PROGRAM P2_06_Device_Ctrl
VAR
	
	fbDischargeValve				:FB_Valve53_Ctrl;	
	bDischargeOpen					:BOOL;
	bDischargeClose					:BOOL;

	fbMixer_Cmd						:FB_Mixer_Ctrl;
	fbMixerSpeed_Cmd				:FB_AnalogOutput;
	fbMixerSpeed_Cmd2				:FB_Scale;

	fChopper1_Cmd					:FB_Chopper_Ctrl;
	fChopper2_Cmd					:FB_Chopper_Ctrl;
	
	fbWater_V1020_Cmd				:FB_Valve_Ctrl;
	fbWarmWater_Cmd					:FB_Valve_Ctrl;
	fbColdWater_Cmd					:FB_Valve_Ctrl;
	fbProcessWater_V1025_Cmd		:FB_Valve_Ctrl;
	fbCleaningAir_V1030_Cmd			:FB_Valve_Ctrl;
	fbTightAir_V1100_Cmd			:FB_Valve_Ctrl;
	
	fbChopper1_Air_V1080_Cmd		:FB_Valve_Ctrl;
	fbChopper1_Water_V1580_Cmd		:FB_Valve_Ctrl;
	fbChopper1_Drain_V1150_Cmd		:FB_Valve_Ctrl;
	
	fbChopper2_Air_V1090_Cmd		:FB_Valve_Ctrl;
	fbChopper2_Water_V1570_Cmd		:FB_Valve_Ctrl;
	fbChopper2_Drain_V1160_Cmd		:FB_Valve_Ctrl;
	
	fbDrainSocket_V1010_Cmd			:FB_Valve_Ctrl;
	
	tonChopper2Delay				:TON;
	
	test		:BOOL;
	fbMixerSpeed_Cmd3: FB_Scale;
	TON_0: TON;
	TON_1: TON;
	TON_2: TON;
END_VAR

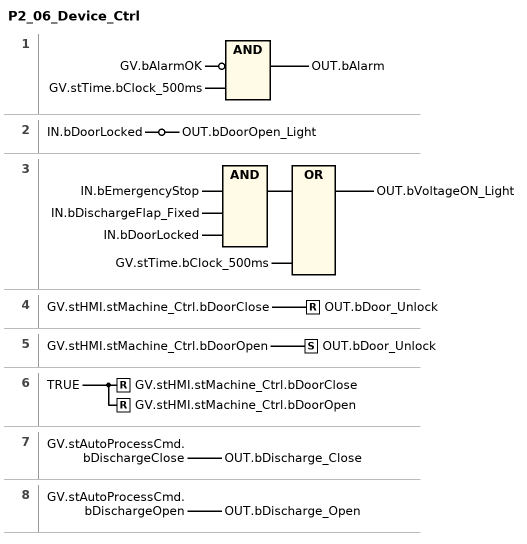
// NETWORK 1
OUT.bAlarm := NOT GV.bAlarmOK AND GV.stTime.bClock_500ms;

// NETWORK 2
OUT.bDoorOpen_Light := NOT IN.bDoorLocked;

// NETWORK 3
OUT.bVoltageON_Light := IN.bEmergencyStop AND IN.bDischargeFlap_Fixed AND IN.bDoorLocked OR GV.stTime.bClock_500ms;

// NETWORK 4
OUT.bDoor_Unlock R= GV.stHMI.stMachine_Ctrl.bDoorClose;

// NETWORK 5
OUT.bDoor_Unlock S= GV.stHMI.stMachine_Ctrl.bDoorOpen;

// NETWORK 6
GV.stHMI.stMachine_Ctrl.bDoorClose R= TRUE;
GV.stHMI.stMachine_Ctrl.bDoorOpen R= TRUE;

// NETWORK 7
OUT.bDischarge_Close := GV.stAutoProcessCmd.bDischargeClose;

// NETWORK 8
OUT.bDischarge_Open := GV.stAutoProcessCmd.bDischargeOpen;

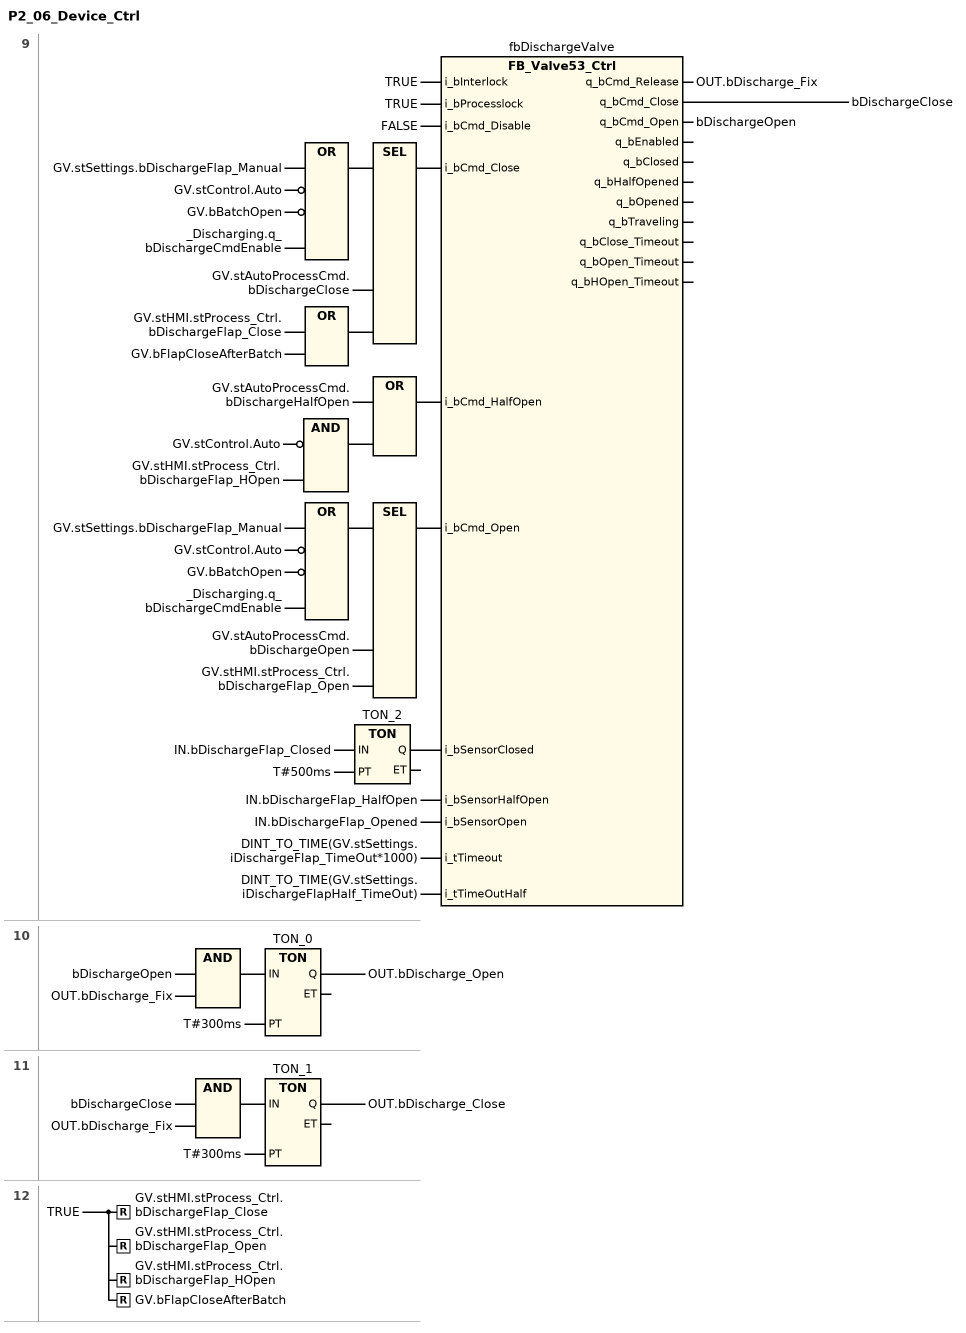
// NETWORK 9
TON_2(IN := IN.bDischargeFlap_Closed, PT := T#500ms); // TON
fbDischargeValve(
    i_bInterlock := TRUE,
    i_bProcesslock := TRUE,
    i_bCmd_Disable := FALSE,
    i_bCmd_Close := SEL(GV.stSettings.bDischargeFlap_Manual OR NOT GV.stControl.Auto OR NOT GV.bBatchOpen OR _Discharging.q_bDischargeCmdEnable, GV.stAutoProcessCmd.bDischargeClose, GV.stHMI.stProcess_Ctrl.bDischargeFlap_Close OR GV.bFlapCloseAfterBatch),
    i_bCmd_HalfOpen := GV.stAutoProcessCmd.bDischargeHalfOpen OR NOT GV.stControl.Auto AND GV.stHMI.stProcess_Ctrl.bDischargeFlap_HOpen,
    i_bCmd_Open := SEL(GV.stSettings.bDischargeFlap_Manual OR NOT GV.stControl.Auto OR NOT GV.bBatchOpen OR _Discharging.q_bDischargeCmdEnable, GV.stAutoProcessCmd.bDischargeOpen, GV.stHMI.stProcess_Ctrl.bDischargeFlap_Open),
    i_bSensorClosed := TON_2.Q,
    i_bSensorHalfOpen := IN.bDischargeFlap_HalfOpen,
    i_bSensorOpen := IN.bDischargeFlap_Opened,
    i_tTimeout := DINT_TO_TIME(GV.stSettings.iDischargeFlap_TimeOut*1000),
    i_tTimeOutHalf := DINT_TO_TIME(GV.stSettings.iDischargeFlapHalf_TimeOut),
    q_bCmd_Release => OUT.bDischarge_Fix,
    q_bCmd_Open => bDischargeOpen); // FB_Valve53_Ctrl
bDischargeClose := fbDischargeValve.q_bCmd_Close;

// NETWORK 10
TON_0(IN := bDischargeOpen AND OUT.bDischarge_Fix, PT := T#300ms); // TON
OUT.bDischarge_Open := TON_0.Q;

// NETWORK 11
TON_1(IN := bDischargeClose AND OUT.bDischarge_Fix, PT := T#300ms); // TON
OUT.bDischarge_Close := TON_1.Q;

// NETWORK 12
GV.stHMI.stProcess_Ctrl.bDischargeFlap_Close R= TRUE;
GV.stHMI.stProcess_Ctrl.bDischargeFlap_Open R= TRUE;
GV.stHMI.stProcess_Ctrl.bDischargeFlap_HOpen R= TRUE;
GV.bFlapCloseAfterBatch R= TRUE;

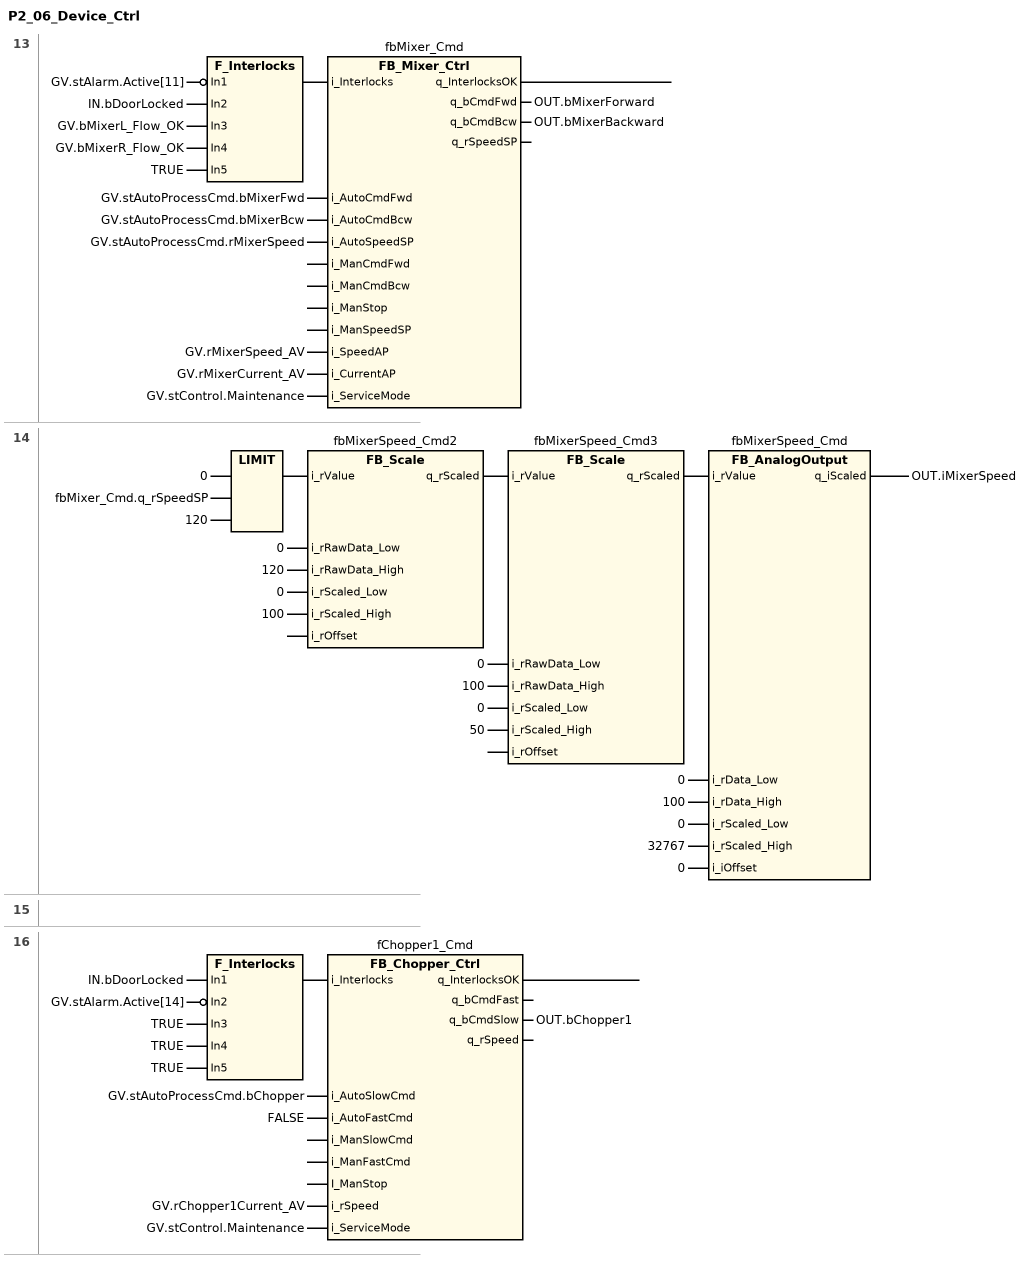
// NETWORK 13
fbMixer_Cmd(
    i_Interlocks := F_Interlocks(In1 := NOT GV.stAlarm.Active[11], In2 := IN.bDoorLocked, In3 := GV.bMixerL_Flow_OK, In4 := GV.bMixerR_Flow_OK, In5 := TRUE),
    i_AutoCmdFwd := GV.stAutoProcessCmd.bMixerFwd,
    i_AutoCmdBcw := GV.stAutoProcessCmd.bMixerBcw,
    i_AutoSpeedSP := GV.stAutoProcessCmd.rMixerSpeed,
    i_SpeedAP := GV.rMixerSpeed_AV,
    i_CurrentAP := GV.rMixerCurrent_AV,
    i_ServiceMode := GV.stControl.Maintenance,
    q_bCmdFwd => OUT.bMixerForward,
    q_bCmdBcw => OUT.bMixerBackward); // FB_Mixer_Ctrl

// NETWORK 14
fbMixerSpeed_Cmd2(
    i_rValue := LIMIT(0, fbMixer_Cmd.q_rSpeedSP, 120),
    i_rRawData_Low := 0,
    i_rRawData_High := 120,
    i_rScaled_Low := 0,
    i_rScaled_High := 100); // FB_Scale
fbMixerSpeed_Cmd3(
    i_rValue := fbMixerSpeed_Cmd2.q_rScaled,
    i_rRawData_Low := 0,
    i_rRawData_High := 100,
    i_rScaled_Low := 0,
    i_rScaled_High := 50); // FB_Scale
fbMixerSpeed_Cmd(
    i_rValue := fbMixerSpeed_Cmd3.q_rScaled,
    i_rData_Low := 0,
    i_rData_High := 100,
    i_rScaled_Low := 0,
    i_rScaled_High := 32767,
    i_iOffset := 0); // FB_AnalogOutput
OUT.iMixerSpeed := fbMixerSpeed_Cmd.q_iScaled;

// NETWORK 15

// NETWORK 16
fChopper1_Cmd(
    i_Interlocks := F_Interlocks(In1 := IN.bDoorLocked, In2 := NOT GV.stAlarm.Active[14], In3 := TRUE, In4 := TRUE, In5 := TRUE),
    i_AutoSlowCmd := GV.stAutoProcessCmd.bChopper,
    i_AutoFastCmd := FALSE,
    i_rSpeed := GV.rChopper1Current_AV,
    i_ServiceMode := GV.stControl.Maintenance,
    q_bCmdSlow => OUT.bChopper1); // FB_Chopper_Ctrl

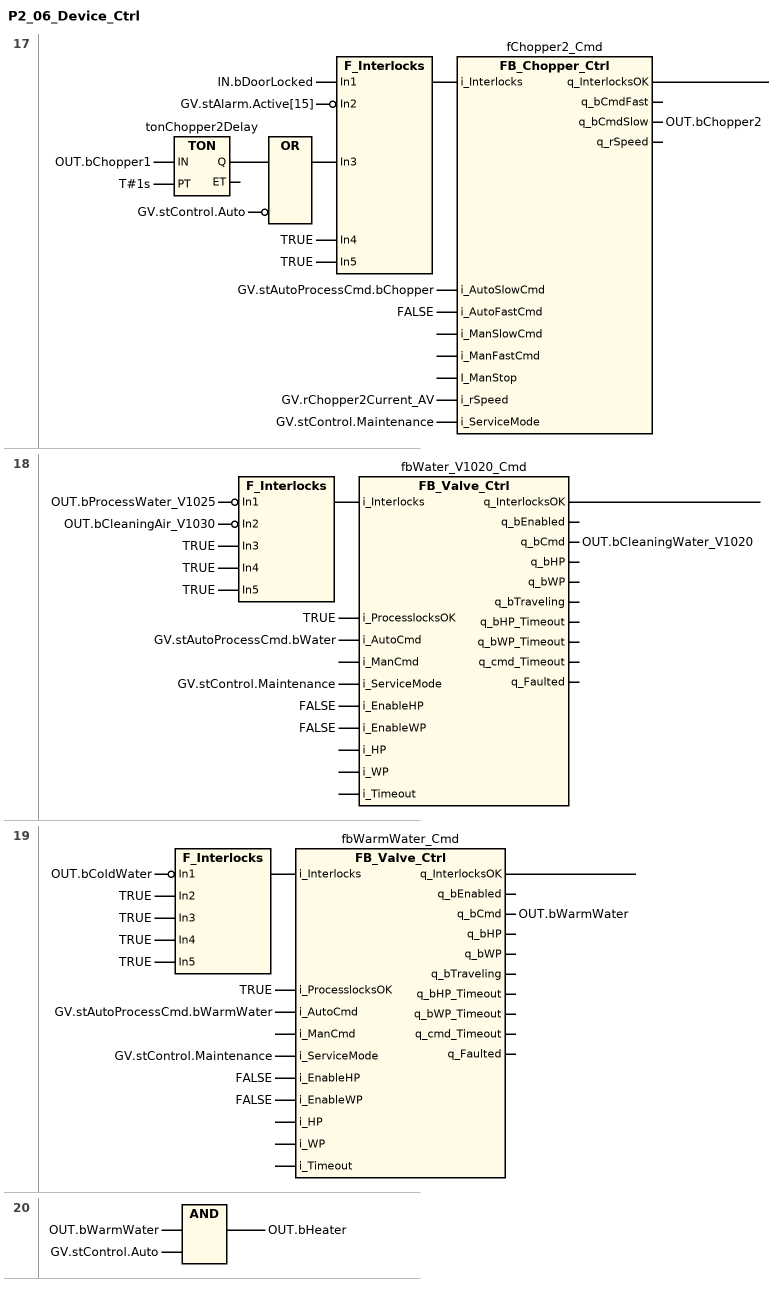
// NETWORK 17
tonChopper2Delay(IN := OUT.bChopper1, PT := T#1s); // TON
fChopper2_Cmd(
    i_Interlocks := F_Interlocks(In1 := IN.bDoorLocked, In2 := NOT GV.stAlarm.Active[15], In3 := tonChopper2Delay.Q OR NOT GV.stControl.Auto, In4 := TRUE, In5 := TRUE),
    i_AutoSlowCmd := GV.stAutoProcessCmd.bChopper,
    i_AutoFastCmd := FALSE,
    i_rSpeed := GV.rChopper2Current_AV,
    i_ServiceMode := GV.stControl.Maintenance,
    q_bCmdSlow => OUT.bChopper2); // FB_Chopper_Ctrl

// NETWORK 18
fbWater_V1020_Cmd(
    i_Interlocks := F_Interlocks(In1 := NOT OUT.bProcessWater_V1025, In2 := NOT OUT.bCleaningAir_V1030, In3 := TRUE, In4 := TRUE, In5 := TRUE),
    i_ProcesslocksOK := TRUE,
    i_AutoCmd := GV.stAutoProcessCmd.bWater,
    i_ServiceMode := GV.stControl.Maintenance,
    i_EnableHP := FALSE,
    i_EnableWP := FALSE,
    q_bCmd => OUT.bCleaningWater_V1020); // FB_Valve_Ctrl

// NETWORK 19
fbWarmWater_Cmd(
    i_Interlocks := F_Interlocks(In1 := NOT OUT.bColdWater, In2 := TRUE, In3 := TRUE, In4 := TRUE, In5 := TRUE),
    i_ProcesslocksOK := TRUE,
    i_AutoCmd := GV.stAutoProcessCmd.bWarmWater,
    i_ServiceMode := GV.stControl.Maintenance,
    i_EnableHP := FALSE,
    i_EnableWP := FALSE,
    q_bCmd => OUT.bWarmWater); // FB_Valve_Ctrl

// NETWORK 20
OUT.bHeater := OUT.bWarmWater AND GV.stControl.Auto;

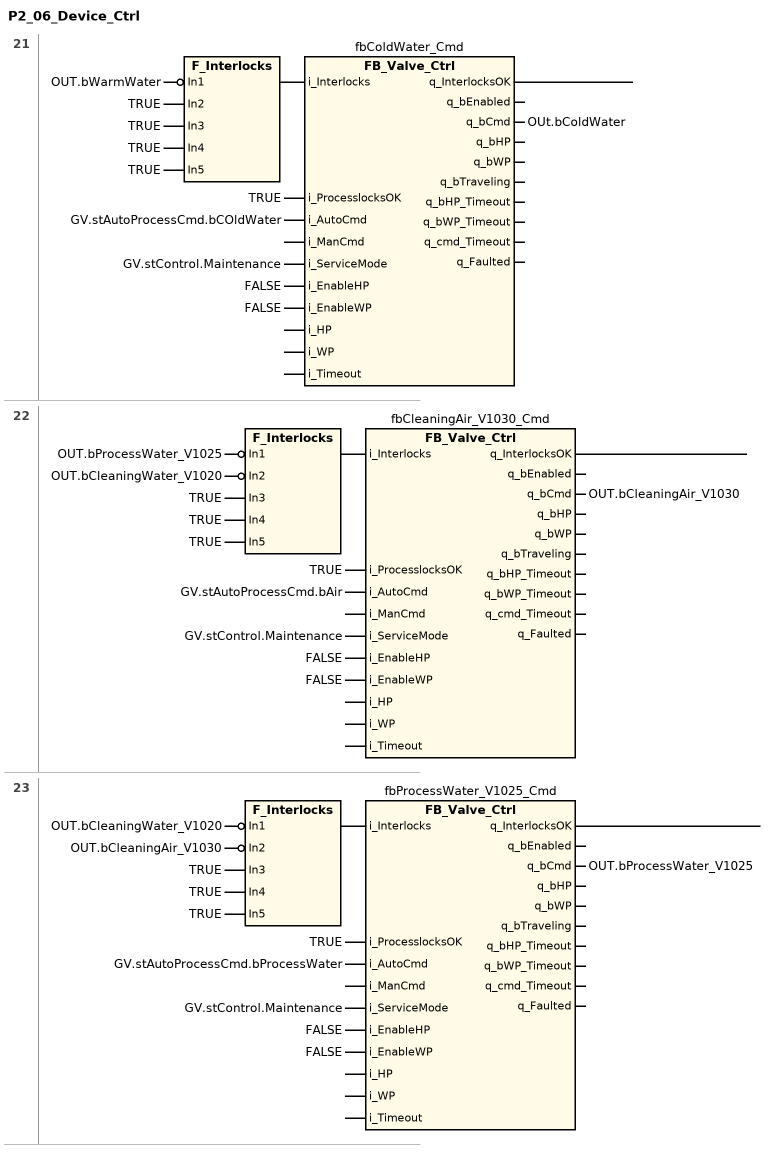
// NETWORK 21
fbColdWater_Cmd(
    i_Interlocks := F_Interlocks(In1 := NOT OUT.bWarmWater, In2 := TRUE, In3 := TRUE, In4 := TRUE, In5 := TRUE),
    i_ProcesslocksOK := TRUE,
    i_AutoCmd := GV.stAutoProcessCmd.bCOldWater,
    i_ServiceMode := GV.stControl.Maintenance,
    i_EnableHP := FALSE,
    i_EnableWP := FALSE,
    q_bCmd => OUt.bColdWater); // FB_Valve_Ctrl

// NETWORK 22
fbCleaningAir_V1030_Cmd(
    i_Interlocks := F_Interlocks(In1 := NOT OUT.bProcessWater_V1025, In2 := NOT OUT.bCleaningWater_V1020, In3 := TRUE, In4 := TRUE, In5 := TRUE),
    i_ProcesslocksOK := TRUE,
    i_AutoCmd := GV.stAutoProcessCmd.bAir,
    i_ServiceMode := GV.stControl.Maintenance,
    i_EnableHP := FALSE,
    i_EnableWP := FALSE,
    q_bCmd => OUT.bCleaningAir_V1030); // FB_Valve_Ctrl

// NETWORK 23
fbProcessWater_V1025_Cmd(
    i_Interlocks := F_Interlocks(In1 := NOT OUT.bCleaningWater_V1020, In2 := NOT OUT.bCleaningAir_V1030, In3 := TRUE, In4 := TRUE, In5 := TRUE),
    i_ProcesslocksOK := TRUE,
    i_AutoCmd := GV.stAutoProcessCmd.bProcessWater,
    i_ServiceMode := GV.stControl.Maintenance,
    i_EnableHP := FALSE,
    i_EnableWP := FALSE,
    q_bCmd => OUT.bProcessWater_V1025); // FB_Valve_Ctrl

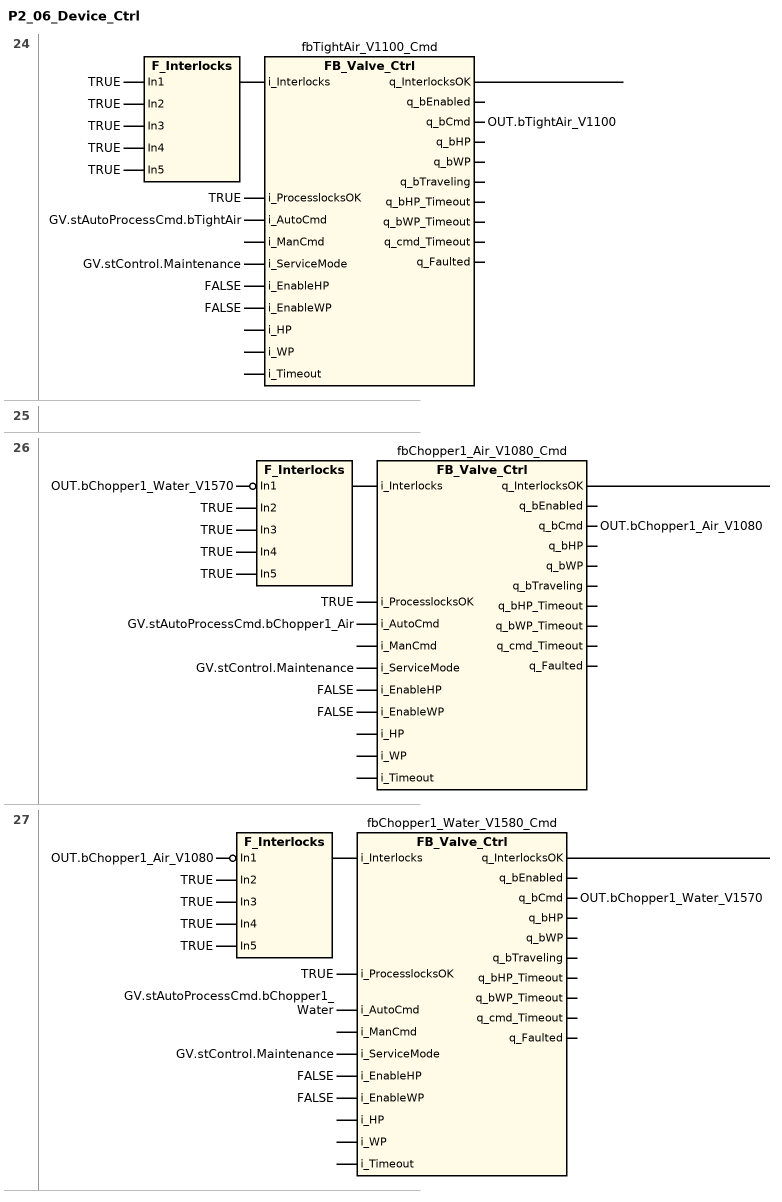
// NETWORK 24
fbTightAir_V1100_Cmd(
    i_Interlocks := F_Interlocks(In1 := TRUE, In2 := TRUE, In3 := TRUE, In4 := TRUE, In5 := TRUE),
    i_ProcesslocksOK := TRUE,
    i_AutoCmd := GV.stAutoProcessCmd.bTightAir,
    i_ServiceMode := GV.stControl.Maintenance,
    i_EnableHP := FALSE,
    i_EnableWP := FALSE,
    q_bCmd => OUT.bTightAir_V1100); // FB_Valve_Ctrl

// NETWORK 25

// NETWORK 26
fbChopper1_Air_V1080_Cmd(
    i_Interlocks := F_Interlocks(In1 := NOT OUT.bChopper1_Water_V1570, In2 := TRUE, In3 := TRUE, In4 := TRUE, In5 := TRUE),
    i_ProcesslocksOK := TRUE,
    i_AutoCmd := GV.stAutoProcessCmd.bChopper1_Air,
    i_ServiceMode := GV.stControl.Maintenance,
    i_EnableHP := FALSE,
    i_EnableWP := FALSE,
    q_bCmd => OUT.bChopper1_Air_V1080); // FB_Valve_Ctrl

// NETWORK 27
fbChopper1_Water_V1580_Cmd(
    i_Interlocks := F_Interlocks(In1 := NOT OUT.bChopper1_Air_V1080, In2 := TRUE, In3 := TRUE, In4 := TRUE, In5 := TRUE),
    i_ProcesslocksOK := TRUE,
    i_AutoCmd := GV.stAutoProcessCmd.bChopper1_Water,
    i_ServiceMode := GV.stControl.Maintenance,
    i_EnableHP := FALSE,
    i_EnableWP := FALSE,
    q_bCmd => OUT.bChopper1_Water_V1570); // FB_Valve_Ctrl

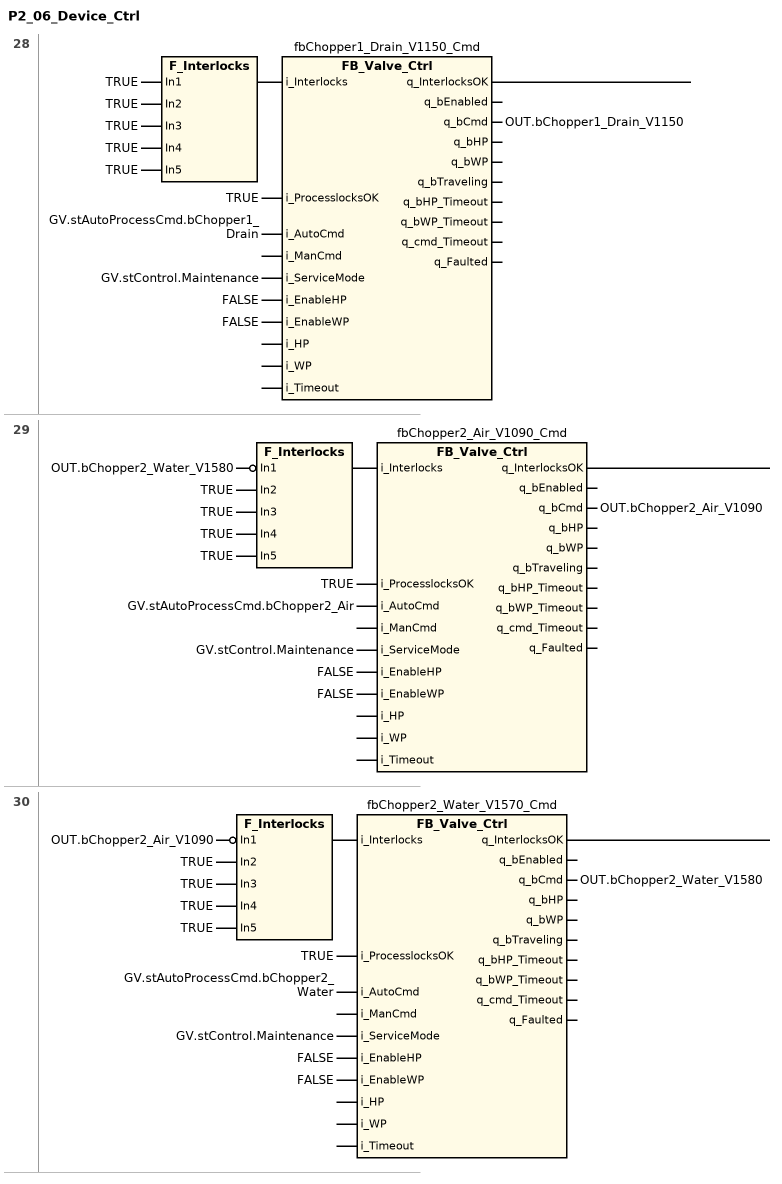
// NETWORK 28
fbChopper1_Drain_V1150_Cmd(
    i_Interlocks := F_Interlocks(In1 := TRUE, In2 := TRUE, In3 := TRUE, In4 := TRUE, In5 := TRUE),
    i_ProcesslocksOK := TRUE,
    i_AutoCmd := GV.stAutoProcessCmd.bChopper1_Drain,
    i_ServiceMode := GV.stControl.Maintenance,
    i_EnableHP := FALSE,
    i_EnableWP := FALSE,
    q_bCmd => OUT.bChopper1_Drain_V1150); // FB_Valve_Ctrl

// NETWORK 29
fbChopper2_Air_V1090_Cmd(
    i_Interlocks := F_Interlocks(In1 := NOT OUT.bChopper2_Water_V1580, In2 := TRUE, In3 := TRUE, In4 := TRUE, In5 := TRUE),
    i_ProcesslocksOK := TRUE,
    i_AutoCmd := GV.stAutoProcessCmd.bChopper2_Air,
    i_ServiceMode := GV.stControl.Maintenance,
    i_EnableHP := FALSE,
    i_EnableWP := FALSE,
    q_bCmd => OUT.bChopper2_Air_V1090); // FB_Valve_Ctrl

// NETWORK 30
fbChopper2_Water_V1570_Cmd(
    i_Interlocks := F_Interlocks(In1 := NOT OUT.bChopper2_Air_V1090, In2 := TRUE, In3 := TRUE, In4 := TRUE, In5 := TRUE),
    i_ProcesslocksOK := TRUE,
    i_AutoCmd := GV.stAutoProcessCmd.bChopper2_Water,
    i_ServiceMode := GV.stControl.Maintenance,
    i_EnableHP := FALSE,
    i_EnableWP := FALSE,
    q_bCmd => OUT.bChopper2_Water_V1580); // FB_Valve_Ctrl

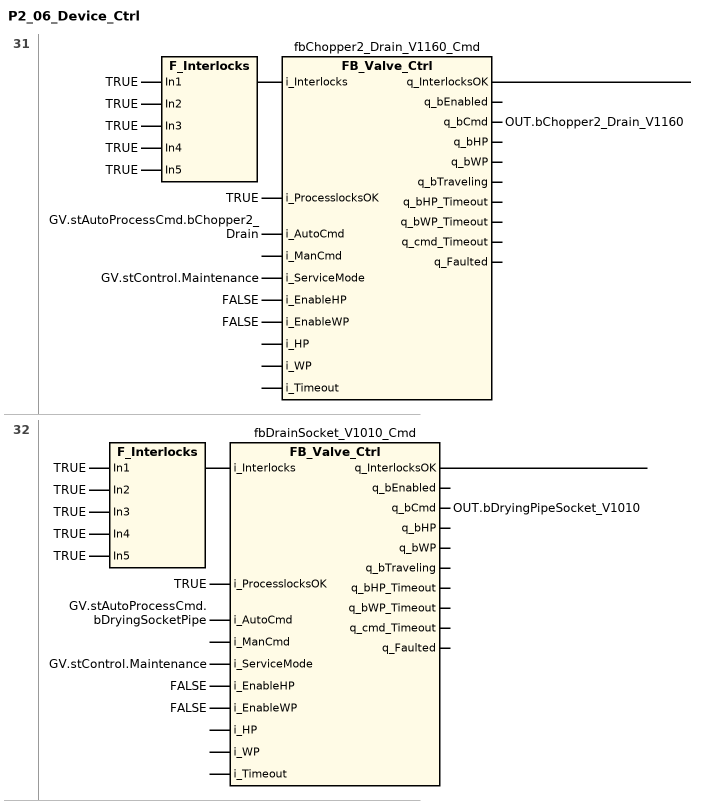
// NETWORK 31
fbChopper2_Drain_V1160_Cmd(
    i_Interlocks := F_Interlocks(In1 := TRUE, In2 := TRUE, In3 := TRUE, In4 := TRUE, In5 := TRUE),
    i_ProcesslocksOK := TRUE,
    i_AutoCmd := GV.stAutoProcessCmd.bChopper2_Drain,
    i_ServiceMode := GV.stControl.Maintenance,
    i_EnableHP := FALSE,
    i_EnableWP := FALSE,
    q_bCmd => OUT.bChopper2_Drain_V1160); // FB_Valve_Ctrl

// NETWORK 32
fbDrainSocket_V1010_Cmd(
    i_Interlocks := F_Interlocks(In1 := TRUE, In2 := TRUE, In3 := TRUE, In4 := TRUE, In5 := TRUE),
    i_ProcesslocksOK := TRUE,
    i_AutoCmd := GV.stAutoProcessCmd.bDryingSocketPipe,
    i_ServiceMode := GV.stControl.Maintenance,
    i_EnableHP := FALSE,
    i_EnableWP := FALSE,
    q_bCmd => OUT.bDryingPipeSocket_V1010); // FB_Valve_Ctrl

END_PROGRAM

(* stored: Version 1.1.0.1
   POU P2_06_Device_Ctrl: Id {a0f0b33c-ae51-440e-85bb-a2c6067bd1da}, SpecialFunc None *)
